TYPE ST_TCPIP_AddressPort :
STRUCT
	IP			: T_IPv4Addr;
	Port		: UINT;
END_STRUCT
END_TYPE

(* stored: Version 1.1.0.1, ProductVersion 3.1.4024.15
   DUT ST_TCPIP_AddressPort: Id {2b3009af-55c9-4f82-9693-7de329701810} *)
